TYPE Router_Standard :
STRUCT
		MesData				: Router ;  (* Object *)

		
END_STRUCT
END_TYPE

(* stored: Version 1.1.0.1, ProductVersion 3.1.4024.6
   DUT Router_Standard: Id {ddf0ced3-74e7-42e5-a40e-84d8a20f5710} *)
